(* IEC 61131-3 sources: SafePLC-Gen-Evaluation/Evaluation Results/P_ID/run_05, 2 files *)

(* ---- io_declarations.st ---- *)
(* ==================================================  *)
(* PLC I/O Variable Declarations — CODESYS 3.5  *)
(* Generated by SafePLC-Gen Multimodal  *)
(* ==================================================  *)

VAR_GLOBAL
    (* --- Analog Inputs ---  *)
    FT_10_Raw                    AT %IW0       : INT := 0;    (* FT-10 — Flow transmitter on upper process line b  *)
    FT_11_Raw                    AT %IW2       : INT := 0;    (* FT-11 — Flow transmitter on lower process line b  *)
    (* --- Analog Outputs ---  *)
    Fv_3_3040_Out                AT %QW0       : INT := 0;    (* Fv-3-3040 — Flow control valve on upper feed line (f  *)
    Fv_3_3041_Out                AT %QW2       : INT := 0;    (* Fv-3-3041 — Flow control valve on lower feed line (f  *)
END_VAR

(* ---- generated_code.st ---- *)
(* Generated by SafePLC-Gen Multimodal — CODESYS 3.5 *)
(* IEC 61131-3 Structured Text *)
(* Date: 2026-04-25T12:51:56.901102 *)

PROGRAM FlowControl

VAR
    FT_10_Raw                    AT %IW0       : INT := 0;
    FT_11_Raw                    AT %IW2       : INT := 0;
    Fv_3_3040_Out                AT %QW0       : INT := 0;
    Fv_3_3041_Out                AT %QW2       : INT := 0;
END_VAR

VAR
    FT_10_Scaled                 : REAL := 0.0;
    FT_11_Scaled                 : REAL := 0.0;

    FT_10_EU_Min                 : REAL := 0.0;
    FT_10_EU_Span                : REAL := 100.0;
    FT_11_EU_Min                 : REAL := 0.0;
    FT_11_EU_Span                : REAL := 100.0;

    FT_10_HH_SP                  : REAL := 90.0;
    FT_10_H_SP                   : REAL := 80.0;
    FT_10_L_SP                   : REAL := 20.0;
    FT_10_LL_SP                  : REAL := 10.0;
    FT_10_Deadband               : REAL := 2.0;

    FT_10_H                      : BOOL := FALSE;
    FT_10_L                      : BOOL := FALSE;
    FT_10_HH_Latch               : SR := (Q1 := FALSE);
    FT_10_LL_Latch               : SR := (Q1 := FALSE);
    FT_10_HH_Ack                 : BOOL := FALSE;
    FT_10_LL_Ack                 : BOOL := FALSE;

    FT_11_HH_SP                  : REAL := 90.0;
    FT_11_H_SP                   : REAL := 80.0;
    FT_11_L_SP                   : REAL := 20.0;
    FT_11_LL_SP                  : REAL := 10.0;
    FT_11_Deadband               : REAL := 2.0;

    FT_11_H                      : BOOL := FALSE;
    FT_11_L                      : BOOL := FALSE;
    FT_11_HH_Latch               : SR := (Q1 := FALSE);
    FT_11_LL_Latch               : SR := (Q1 := FALSE);
    FT_11_HH_Ack                 : BOOL := FALSE;
    FT_11_LL_Ack                 : BOOL := FALSE;

    FIC_3040_SP                  : REAL := 50.0;
    FIC_3040_Kp                  : REAL := 1.2;
    FIC_3040_Ki                  : REAL := 0.05;
    FIC_3040_Error               : REAL := 0.0;
    FIC_3040_Integral            : REAL := 0.0;
    FIC_3040_Output              : REAL := 0.0;

    FIC_3041_SP                  : REAL := 50.0;
    FIC_3041_Kp                  : REAL := 1.2;
    FIC_3041_Ki                  : REAL := 0.05;
    FIC_3041_Error               : REAL := 0.0;
    FIC_3041_Integral            : REAL := 0.0;
    FIC_3041_Output              : REAL := 0.0;

    ISA_SV_001                   : BOOL := FALSE;
    ISA_SV_002                   : BOOL := FALSE;
    CV_3040_BLK                  : BOOL := FALSE;
    CV_3041_BLK                  : BOOL := FALSE;

    System_Alarm                 : BOOL := FALSE;
    FirstScan                    : BOOL := TRUE;
END_VAR

IF FirstScan THEN
    Fv_3_3040_Out     := 6554;
    Fv_3_3041_Out     := 6554;
    ISA_SV_001        := FALSE;
    ISA_SV_002        := FALSE;
    CV_3040_BLK       := FALSE;
    CV_3041_BLK       := FALSE;
    FIC_3040_Integral := 0.0;
    FIC_3041_Integral := 0.0;
    FirstScan         := FALSE;
    RETURN;
END_IF;

FT_10_Scaled := ((INT_TO_REAL(FT_10_Raw) - 6554.0) / (32767.0 - 6554.0)) * FT_10_EU_Span + FT_10_EU_Min;
FT_11_Scaled := ((INT_TO_REAL(FT_11_Raw) - 6554.0) / (32767.0 - 6554.0)) * FT_11_EU_Span + FT_11_EU_Min;

FT_10_HH_Latch(S1 := FT_10_Scaled >= FT_10_HH_SP,
               R  := FT_10_HH_Ack AND (FT_10_Scaled <= (FT_10_HH_SP - FT_10_Deadband)));

IF FT_10_Scaled >= FT_10_H_SP THEN
    FT_10_H := TRUE;
ELSIF FT_10_Scaled <= (FT_10_H_SP - FT_10_Deadband) THEN
    FT_10_H := FALSE;
END_IF;

IF FT_10_Scaled <= FT_10_L_SP THEN
    FT_10_L := TRUE;
ELSIF FT_10_Scaled >= (FT_10_L_SP + FT_10_Deadband) THEN
    FT_10_L := FALSE;
END_IF;

FT_10_LL_Latch(S1 := FT_10_Scaled <= FT_10_LL_SP,
               R  := FT_10_LL_Ack AND (FT_10_Scaled >= (FT_10_LL_SP + FT_10_Deadband)));

FT_11_HH_Latch(S1 := FT_11_Scaled >= FT_11_HH_SP,
               R  := FT_11_HH_Ack AND (FT_11_Scaled <= (FT_11_HH_SP - FT_11_Deadband)));

IF FT_11_Scaled >= FT_11_H_SP THEN
    FT_11_H := TRUE;
ELSIF FT_11_Scaled <= (FT_11_H_SP - FT_11_Deadband) THEN
    FT_11_H := FALSE;
END_IF;

IF FT_11_Scaled <= FT_11_L_SP THEN
    FT_11_L := TRUE;
ELSIF FT_11_Scaled >= (FT_11_L_SP + FT_11_Deadband) THEN
    FT_11_L := FALSE;
END_IF;

FT_11_LL_Latch(S1 := FT_11_Scaled <= FT_11_LL_SP,
               R  := FT_11_LL_Ack AND (FT_11_Scaled >= (FT_11_LL_SP + FT_11_Deadband)));

FIC_3040_Error    := FIC_3040_SP - FT_10_Scaled;
FIC_3040_Integral := FIC_3040_Integral + (FIC_3040_Ki * FIC_3040_Error);
IF FIC_3040_Integral > 100.0 THEN
    FIC_3040_Integral := 100.0;
ELSIF FIC_3040_Integral < 0.0 THEN
    FIC_3040_Integral := 0.0;
END_IF;
FIC_3040_Output := (FIC_3040_Kp * FIC_3040_Error) + FIC_3040_Integral;
IF FIC_3040_Output > 100.0 THEN
    FIC_3040_Output := 100.0;
ELSIF FIC_3040_Output < 0.0 THEN
    FIC_3040_Output := 0.0;
END_IF;
Fv_3_3040_Out := REAL_TO_INT(6554.0 + (FIC_3040_Output / 100.0) * (32767.0 - 6554.0));

FIC_3041_Error    := FIC_3041_SP - FT_11_Scaled;
FIC_3041_Integral := FIC_3041_Integral + (FIC_3041_Ki * FIC_3041_Error);
IF FIC_3041_Integral > 100.0 THEN
    FIC_3041_Integral := 100.0;
ELSIF FIC_3041_Integral < 0.0 THEN
    FIC_3041_Integral := 0.0;
END_IF;
FIC_3041_Output := (FIC_3041_Kp * FIC_3041_Error) + FIC_3041_Integral;
IF FIC_3041_Output > 100.0 THEN
    FIC_3041_Output := 100.0;
ELSIF FIC_3041_Output < 0.0 THEN
    FIC_3041_Output := 0.0;
END_IF;
Fv_3_3041_Out := REAL_TO_INT(6554.0 + (FIC_3041_Output / 100.0) * (32767.0 - 6554.0));

CV_3040_BLK := NOT FT_10_HH_Latch.Q1 AND NOT FT_10_LL_Latch.Q1;
CV_3041_BLK := NOT FT_11_HH_Latch.Q1 AND NOT FT_11_LL_Latch.Q1;
ISA_SV_001  := CV_3040_BLK;
ISA_SV_002  := CV_3041_BLK;

System_Alarm :=
    FT_10_HH_Latch.Q1 OR FT_10_LL_Latch.Q1 OR FT_10_H OR FT_10_L OR
    FT_11_HH_Latch.Q1 OR FT_11_LL_Latch.Q1 OR FT_11_H OR FT_11_L;

END_PROGRAM
